FUNCTION F_OPSTATE : BOOL
VAR_INPUT
	uStateIn: UINT;
END_VAR
VAR
END_VAR

F_OPSTATE := GETBIT32(inVal32 := uStateIn, bitNo := 3);

END_FUNCTION

(* stored: Version 1.1.0.1, ProductVersion 3.1.4024.12
   POU F_OPSTATE: Id {e4a69484-b6cb-4c74-b304-d981704b0ea6}, SpecialFunc None *)
